FUNCTION_BLOCK FB_2_Skill_RoCo EXTENDS FB_1_Skill
VAR_INPUT
	{attribute 'OPC.UA.DA.StructuredType':=1}
	{attribute 'OPC.UA.DA' := '1'}
	Control     : ST_SkillControl;
	{attribute 'OPC.UA.DA.StructuredType':=1}
	{attribute 'OPC.UA.DA' := '1'}
    Status      : ST_SkillStatus;
END_VAR
VAR_OUTPUT
END_VAR
VAR
// 	SubSkillHandler : FB_SkillHandler;
END_VAR

ACTION CYCLIC_RoCo:
CYCLIC_SKILL();
END_ACTION

METHOD PROTECTED onActivate : eResult
VAR_INPUT
END_VAR

VAR
	eParentResult: eResult;
	myResult: ERESULT;
END_VAR

VAR //YOUR CODE
	succ : BOOL;
END_VAR
eParentResult := SUPER^.onActivate();
//--------------------------------------------------
myResult:=NONE;
// ----- YOUR CODE HERE (incl. Alarms) -------------



// ----- END YOUR CODE -----------------------------
//--------------------------------------------------
onActivate := CombineResults(eParentResult,myResult);
END_METHOD

METHOD PROTECTED onCleanup : eResult
VAR_INPUT
END_VAR

VAR
	eParentResult: eResult;
	myResult: ERESULT;
END_VAR

VAR //YOUR CODE
	succ : BOOL;
END_VAR
eParentResult := SUPER^.onCleanup();
//--------------------------------------------------
myResult:=NONE;
// ----- YOUR CODE HERE (incl. Alarms) -------------



// ----- END YOUR CODE -----------------------------
//--------------------------------------------------
onCleanup := CombineResults(eParentResult,myResult);
END_METHOD

METHOD PROTECTED onConfigure : eResult
VAR_INPUT
END_VAR

VAR
	eParentResult: eResult;
	myResult: ERESULT;
END_VAR

VAR //YOUR CODE
	succ : BOOL;
END_VAR
eParentResult := SUPER^.onConfigure();
//--------------------------------------------------
myResult:=NONE;
// ----- YOUR CODE HERE (incl. Alarms) -------------



// ----- END YOUR CODE -----------------------------
//--------------------------------------------------
onConfigure := CombineResults(eParentResult,myResult);
END_METHOD

METHOD PROTECTED onDeactivate : eResult
VAR_INPUT
END_VAR

VAR
	eParentResult: eResult;
	myResult: ERESULT;
END_VAR

VAR //YOUR CODE
	succ : BOOL;
END_VAR
eParentResult := SUPER^.onDeactivate();
//--------------------------------------------------
myResult:=NONE;
// ----- YOUR CODE HERE (incl. Alarms) -------------



// ----- END YOUR CODE -----------------------------
//--------------------------------------------------
onDeactivate := CombineResults(eParentResult,myResult);
END_METHOD

METHOD PROTECTED onError : eResult
VAR_INPUT
END_VAR

VAR
	eParentResult: eResult;
	myResult: ERESULT;
END_VAR

VAR //YOUR CODE
	succ : BOOL;
END_VAR
eParentResult := SUPER^.onError();
//--------------------------------------------------
myResult:=NONE;
// ----- YOUR CODE HERE (incl. Alarms) -------------



// ----- END YOUR CODE -----------------------------
//--------------------------------------------------
onError := CombineResults(eParentResult,myResult);
END_METHOD

METHOD PROTECTED onShutdown : eResult
VAR_INPUT
END_VAR

VAR
	eParentResult: eResult;
	myResult: ERESULT;
END_VAR

VAR //YOUR CODE
	succ : BOOL;
END_VAR
eParentResult := SUPER^.onShutdown();
//--------------------------------------------------
myResult:=NONE;
// ----- YOUR CODE HERE (incl. Alarms) -------------



// ----- END YOUR CODE -----------------------------
//--------------------------------------------------
onShutdown := CombineResults(eParentResult,myResult);
END_METHOD

END_FUNCTION_BLOCK

(* stored: Version 1.1.0.1, ProductVersion 3.1.4026.18
   POU FB_2_Skill_RoCo: Id {0c991693-7acc-44da-a33b-921e12b69bcf}, SpecialFunc None
   Folder StateControl: Id {dfdaae60-212a-4ac2-b541-e49920b50ee5}
   Action CYCLIC_RoCo: Id {c041a816-ff49-48ac-a22a-009900b81048}
   Method onActivate: Id {646f78db-c383-4e57-9a88-cf5c76b8d7d7}
   Method onCleanup: Id {d57eed92-e820-47f8-9edd-8ec84cb3de8a}
   Method onConfigure: Id {2ca615dc-5172-4946-bb22-b2a7f1793b8a}
   Method onDeactivate: Id {9d819dc0-0217-4955-97fc-efc7b8f817d6}
   Method onError: Id {66d19cc0-3e00-44ec-85bb-a19ef2ca138a}
   Method onShutdown: Id {c6913cb3-7507-4481-9ac7-152b3862865f} *)
